// TIA Portal V17 export
VAR_GLOBAL   // PLC tag table "Safety"
   FaultOk AT %I0.4 : Bool;   // Safety chain feedback OK
END_VAR
